FUNCTION_BLOCK FB_McAxis
VAR
  _AxisRef                      : POINTER TO Tc2_MC2.AXIS_REF;
  _pCalibrationCam              : POINTER TO BOOL;

  _nErrorId                     : UDINT; // datafield for MC error

  // MC_Power inputs for feed fwd, feed bwd, override
  _bEnablePositive              : BOOL  := TRUE;
  _bEnableNegative              : BOOL  := TRUE;
  _rAxisOverride                : LREAL := 100.0;

  _rValueParameterRead          : LREAL;
  _fbReadParameter              : Tc2_MC2.MC_ReadParameter;
  _fbWriteParameter             : Tc2_MC2.MC_WriteParameter;
  _fbWriteParameterPersist      : Tc2_MC2.MC_WriteParameterPersistent;


  // name and encoder type are read by ADSREAD instance from NC
  _sAxisName                    : STRING(30) := 'NO NAME'; // AxisName is limited to 30 chars, IdxGrp := 4000 + _AxisRef.NcToPlc.AxisId, IdxOffs := 16#02
  _sEncoderType                 : STRING(30) := 'NO TYPE';
  _nEncoderType                 : UDINT;
  _eEncoderType                 : E_AxisEncoderType;

  // Motion Control FB Instances
  _fbPower                      : Tc2_MC2.MC_Power;
  _fbReset                      : Tc2_MC2.MC_Reset;
  _fbHalt                       : Tc2_MC2.MC_Halt;
  _fbStop                       : Tc2_MC2.MC_Stop;
  _fbHome                       : Tc2_MC2.MC_Home;
  _fbJog                        : Tc2_MC2.MC_Jog;

  _fbMoveVelocity               : ARRAY[1..2]   OF  Tc2_MC2.MC_MoveVelocity;
  _fbMoveAbsolute               : ARRAY[1..2]   OF  Tc2_MC2.MC_MoveAbsolute;

  // ADS read instance for reading startup information from NC
  _fbADSRead                     : ADSREAD;

  // startup states for getting ADS information from NC
  _nStartUpErrorState,
  _nStartUp                     : DINT := 0;

  _bStartUpError,
  _bStartUp                     : BOOL;

  _rCycleTime                   : LREAL;
  _fbGetCurTaskIndex            : Tc2_System.GETCURTASKINDEX;
END_VAR

PROPERTY AxisEnableNegative : BOOL
GET
AxisEnableNegative := _bEnableNegative;
END_GET
SET
_bEnableNegative := AxisEnableNegative;
END_SET
END_PROPERTY

PROPERTY AxisEnablePositive : BOOL
GET
AxisEnablePositive  := _bEnablePositive;
END_GET
SET
_bEnablePositive := AxisEnablePositive;
END_SET
END_PROPERTY

PROPERTY AxisName : string(30)
GET
AxisName := _sAxisName;
END_GET
END_PROPERTY

PROPERTY AxisRef : pointer to Tc2_MC2.AXIS_REF
SET
_AxisRef := AxisRef;
END_SET
END_PROPERTY

PROPERTY CalibrationCam : pointer to bool
GET
CalibrationCam  := _pCalibrationCam;
END_GET
SET
_pCalibrationCam := CalibrationCam;
END_SET
END_PROPERTY

METHOD Cycle : E_PROGRESS
VAR_INST
  _eState           : E_PROGRESS;
  _rValue           : LREAL;
  _nErrorId         : UDINT;
  _stMsg            : ST_Message;
END_VAR
// call cyclic NC interface
_AxisRef^();

_fbPower(
        Axis                      := _AxisRef^, 
        Enable_Positive           := _bEnablePositive, 
        Enable_Negative           := _bEnableNegative, 
        Override                  := _rAxisOverride);

CASE _eState
OF
  E_PROGRESS.INIT:
    _fbGetCurTaskIndex();
    _rCycleTime                   := UDINT_TO_LREAL(_TaskInfo[_fbGetCurTaskIndex.index].CycleTime)/10000.0;

    _eState                       := E_PROGRESS.BUSY;
END_CASE
CASE _eState
OF
  E_PROGRESS.BUSY:
    IF (_fbPower.Error) OR
       (_AxisRef^.Status.Error)
    THEN
      _eState                     := E_PROGRESS.ERROR;

      _nErrorId                   := SEL((_fbPower.ErrorID > 0), _AxisRef^.NcToPlc.ErrorCode, _fbPower.ErrorID);

      _stMsg.eType                := E_MessageType.eMessageError;
      _stMsg.eDevice              := e_Device.Axis + TO_DINT(_AxisRef^.NcToPlc.AxisId);;
      _stMsg.eSubdevice           := e_Subdevice.fbAxis_Cycle;
      _stMsg.iErrorNumber         := _nErrorId;

      f_MessageSet(_stMsg);
    ELSE
      _nErrorId                   := 0;
      _eState                     := E_PROGRESS.WORKING;
    END_IF
END_CASE
CASE _eState
OF
  E_PROGRESS.WORKING:
    // rinse, repeat
    _eState                       := E_PROGRESS.BUSY;
    Cycle                         := E_PROGRESS.WORKING;
END_CASE
CASE _eState
OF
  E_PROGRESS.ERROR:
    IF NOT (_fbPower.Error)
    THEN
      _eState                     := E_PROGRESS.BUSY;
    ELSE
      Cycle                       := E_PROGRESS.ERROR;
    END_IF
END_CASE
END_METHOD

METHOD Disable : E_PROGRESS
VAR_INPUT
  Execute           : BOOL;
END_VAR
VAR_INST
  _eState           : E_PROGRESS;
  _rValue           : LREAL;
  _stMsg            : ST_Message;


END_VAR
IF NOT Execute THEN _eState := E_PROGRESS.INIT; END_IF

CASE _eState
OF
  E_PROGRESS.INIT:
    IF Execute 
    THEN
      memset(ADR(_stMsg),0,SIZEOF(_stMsg));
      _nErrorId                     := 0;
      _rValue                       := 0;
      _eState                       := E_PROGRESS.BUSY;
    END_IF
END_CASE
CASE _eState
OF
  E_PROGRESS.BUSY:
    _fbPower.Enable                 := FALSE;
    _eState                         := E_PROGRESS.STARTUP;
END_CASE
CASE _eState
OF
  E_PROGRESS.STARTUP:
    IF _fbPower.Error
    THEN
      _eState                       := E_PROGRESS.ERROR;
    ELSE
      _eState                       := E_PROGRESS.WAITING;
    END_IF
END_CASE
CASE _eState
OF
  E_PROGRESS.WAITING:
    IF _AxisRef^.Status.Error
    THEN
      _nErrorId                     := _AxisRef^.NcToPlc.ErrorCode;
    
      _stMsg.eType                  := E_MessageType.eMessageError;
      _stMsg.eDevice                := e_Device.Axis + TO_DINT(_AxisRef^.NcToPlc.AxisId);
      _stMsg.eSubdevice             :=  e_SubDevice.AxisControl;
      _stMsg.iErrorNumber           := _nErrorId;

      f_MessageSet(_stMsg);
    
      _eState                       := E_PROGRESS.ERROR;

    ELSIF NOT _AxisRef^.Status.ControlLoopClosed
    THEN
      _eState                       := E_PROGRESS.WORKING;
    END_IF
END_CASE
CASE _eState
OF
  E_PROGRESS.WORKING:
    _eState                         := E_PROGRESS.DONE;
END_CASE

Disable := _eState;
END_METHOD

METHOD Enable : E_PROGRESS
VAR_INPUT
  Execute           : BOOL;
END_VAR
VAR_INST
  _eState           : E_PROGRESS;
  _rValue           : LREAL;
  _stMsg            : ST_Message;
END_VAR
IF NOT Execute THEN _eState := E_PROGRESS.INIT; END_IF

CASE _eState
OF
  E_PROGRESS.INIT:
    IF Execute 
    THEN
      memset(ADR(_stMsg),0,SIZEOF(_stMsg));
      _nErrorId                     := 0;
      _rValue                       := 0;
      _eState                       := E_PROGRESS.BUSY;
    END_IF
END_CASE
CASE _eState
OF
  E_PROGRESS.BUSY:
    _fbPower.Enable                 := TRUE;
    _eState                         := E_PROGRESS.STARTUP;
END_CASE
CASE _eState
OF
  E_PROGRESS.STARTUP:
    IF _fbPower.Error
    THEN
      _fbPower.Enable               := FALSE;
      _eState                       := E_PROGRESS.ERROR;
    ELSE
      _eState                       := E_PROGRESS.WAITING;
    END_IF
END_CASE
CASE _eState
OF
  E_PROGRESS.WAITING:
    IF _AxisRef^.Status.Error
    THEN
      _nErrorId                     := _AxisRef^.NcToPlc.ErrorCode;
    
      _stMsg.eType                  := E_MessageType.eMessageError;
      _stMsg.eDevice                := e_Device.Axis + TO_DINT(_AxisRef^.NcToPlc.AxisId);
      _stMsg.eSubdevice             :=  e_SubDevice.AxisControl;
      _stMsg.iErrorNumber           := _nErrorId;
    
      f_MessageSet(_stMsg);

      _eState                       := E_PROGRESS.ERROR;

    ELSIF _AxisRef^.Status.ControlLoopClosed
    THEN
      _eState                       := E_PROGRESS.WORKING;
    END_IF
END_CASE
CASE _eState
OF
  E_PROGRESS.WORKING:
    _eState                         := E_PROGRESS.DONE;
END_CASE

Enable                              := _eState;
END_METHOD

PROPERTY EncoderType : E_AxisEncoderType
GET
EncoderType := _eEncoderType;
END_GET
END_PROPERTY

PROPERTY ErrorId : udint
GET
ErrorId := _nErrorId;
END_GET
END_PROPERTY

METHOD Halt : E_PROGRESS
VAR_INPUT
  Execute           : BOOL;
  Dec               : LREAL;
  Jerk              : LREAL;
END_VAR
VAR_INST
  _eState           : E_PROGRESS;
  _rValue           : LREAL;
  _stMsg            : ST_Message;
END_VAR
IF NOT Execute THEN _eState := E_PROGRESS.INIT; END_IF

CASE _eState
OF
  E_PROGRESS.INIT:
    IF Execute 
    THEN
      memset(ADR(_stMsg),0,SIZEOF(_stMsg));
      _nErrorId                     := 0;
      _rValue                       := 0;
      _eState                       := E_PROGRESS.BUSY;
    END_IF
END_CASE
CASE _eState
OF
  E_PROGRESS.BUSY:
    _eState                         := E_PROGRESS.WAITING;
    _fbHalt(
              Axis                  := _AxisRef^, 
              Execute               := FALSE, 
              Deceleration          := Dec, 
              Jerk                  := Jerk, 
              BufferMode            := Tc2_MC2.MC_BufferMode.MC_Aborting);
END_CASE
CASE _eState
OF
  E_PROGRESS.WAITING:
    _fbHalt(
              Axis                  := _AxisRef^, 
              Execute               := TRUE, 
              Deceleration          := Dec, 
              Jerk                  := Jerk, 
              BufferMode            := Tc2_MC2.MC_BufferMode.MC_Aborting);

    IF _fbhalt.Error
    THEN
        _nErrorId                   := _fbHalt.ErrorID;

        _stMsg.eType                := E_MessageType.eMessageError;
        _stMsg.eDevice              := e_Device.Axis + TO_DINT(_AxisRef^.NcToPlc.AxisId);
        _stMsg.eSubdevice           := e_SubDevice.fbHalt;
        _stMsg.iErrorNumber         := _nErrorId;

        f_MessageSet(_stMsg);
        _fbHalt(
              Axis                  := _AxisRef^, 
              Execute               := FALSE);

      _eState                       := E_PROGRESS.ERROR;

    ELSE
      IF _fbHalt.Done OR
         _AxisRef^.Status.NotMoving
      THEN
        _eState                     := E_PROGRESS.WORKING;

      ELSIF _fbHalt.CommandAborted
      THEN
        _eState                     := E_PROGRESS.BUSY;
      END_IF
    END_IF
END_CASE
CASE _eState
OF
  E_PROGRESS.WORKING:
    _fbHalt(
              Axis                  := _AxisRef^, 
              Execute               := FALSE);

    _eState                         := E_PROGRESS.DONE;
END_CASE

Halt := _eState;
END_METHOD

METHOD Home : E_PROGRESS
VAR_INPUT
  Execute           : BOOL;
  Position          : LREAL := DEFAULT_HOME_POSITION;
  HomingMode        : Tc2_MC2.MC_HomingMode := MC_DefaultHoming;
  Options           : Tc2_MC2.ST_HomingOptions;
END_VAR
VAR_INST
  _eState           : E_PROGRESS;
  _sValue           : STRING(40);
  _rValue           : LREAL;
  _stMsg            : ST_Message;
END_VAR
IF NOT Execute THEN _eState := E_PROGRESS.INIT; END_IF

CASE _eState
OF
  E_PROGRESS.INIT:
    IF Execute 
    THEN
      memset(ADR(_stMsg), 0,SIZEOF(_stMsg));
      memset(ADR(_sValue),0,SIZEOF(_sValue));

      _nErrorId                     := 0;
      _rValue                       := 0;
      _eState                       := E_PROGRESS.BUSY;

      IF NOT (_pCalibrationCam <> 0) 
      THEN
        // prevent page fault
        _sValue                     := 'Pointer to calibration cam not set';

        _nErrorId                   := 666;

        _stMsg.eType                := E_MessageType.eMessageError;
        _stMsg.eDevice              := e_Device.Axis + TO_DINT(_AxisRef^.NcToPlc.AxisId);
        _stMsg.eSubdevice           := e_SubDevice.fbHome;
        _stMsg.iErrorNumber         := _nErrorId;
        _stMsg.sText                := _sValue;

        f_MessageSet(_stMsg);

        _eState                     := E_PROGRESS.ERROR;
      END_IF
    END_IF
END_CASE
CASE _eState
OF
  E_PROGRESS.BUSY:
    _eState                         := E_PROGRESS.WAITING;
    _fbHome(
            Axis                    := _AxisRef^, 
            Execute                 := FALSE, 
            Position                := Position, 
            HomingMode              := HomingMode, 
            Options                 := Options, 
            bCalibrationCam         := _pCalibrationCam^);
END_CASE
CASE _eState
OF
  E_PROGRESS.WAITING:
    _fbHome(
            Execute                 := TRUE, 
            Axis                    := _AxisRef^);

    IF _fbHome.Done
    THEN
      _eState                       := E_PROGRESS.WORKING;
    ELSE
      IF _fbHome.Error
      THEN
        _eState                     := E_PROGRESS.ERROR;
        _nErrorId                   := _fbHome.ErrorID;

        _stMsg.eType                := E_MessageType.eMessageError;
        _stMsg.eDevice              := e_Device.Axis + TO_DINT(_AxisRef^.NcToPlc.AxisId);
        _stMsg.eSubdevice           :=  e_SubDevice.fbHome;
        _stMsg.iErrorNumber         := _nErrorId;

        f_MessageSet(_stMsg);

        _fbHome(
            Execute                 := FALSE, 
            Axis                    := _AxisRef^);
      END_IF
    END_IF
END_CASE
CASE _eState
OF
  E_PROGRESS.WORKING:
    _fbHome(
            Execute                 := FALSE, 
            Axis                    := _AxisRef^);

    _eState                         := E_PROGRESS.DONE;
END_CASE

Home                                := _eState;
END_METHOD

METHOD MovePosBuffer : E_PROGRESS
VAR_INPUT
  Enable          : BOOL;
  Position        : LREAL;
  Vel             : LREAL;
  Acc             : LREAL;
  Dec             : LREAL;
  Jerk            : LREAL;
  BufferMode      : Tc2_MC2.MC_BufferMode;
END_VAR
VAR_INST
  _eState           : E_PROGRESS;
  _rValue           : LREAL;
  _stMsg            : ST_Message;
END_VAR
IF NOT Enable THEN _eState := E_PROGRESS.INIT; END_IF

CASE _eState
OF
  E_PROGRESS.INIT:
    IF Enable 
    THEN
      memset(ADR(_stMsg),0,SIZEOF(_stMsg));
      _nErrorId                     := 0;
      _rValue                       := 0;
      _eState                       := E_PROGRESS.BUSY;
    END_IF
END_CASE
CASE _eState
OF
  E_PROGRESS.BUSY:
    _eState                         := E_PROGRESS.STARTUP;
    _rValue                         := Position;

    _fbMoveAbsolute[1](Axis         := _AxisRef^,
                       Execute      := FALSE);
    _fbMoveAbsolute[2](Axis         := _AxisRef^,
                       Execute      := FALSE);

END_CASE
CASE _eState
OF
  E_PROGRESS.STARTUP:
    _fbMoveAbsolute[1](
                    Axis            := _AxisRef^, 
                    Execute         := TRUE,
                    Position        := _rValue, 
                    Velocity        := Vel, 
                    Acceleration    := Acc, 
                    Deceleration    := Dec, 
                    Jerk            := Jerk, 
                    BufferMode      := BufferMode);

    _fbMoveAbsolute[2](
                    Axis            := _AxisRef^, 
                    Execute         := FALSE, 
                    Velocity        := Vel, 
                    Acceleration    := Acc, 
                    Deceleration    := Dec, 
                    Jerk            := Jerk, 
                    BufferMode      := BufferMode);

    _eState                         := E_PROGRESS.PREPARE;
END_CASE
CASE _eState
OF
  E_PROGRESS.PREPARE:
    _fbMoveAbsolute[1](Axis         := _AxisRef^);
    _fbMoveAbsolute[2](Axis         := _AxisRef^);

    IF (Position <> _rValue)
    THEN
      _rValue                       := Position;
      _eState                       := E_PROGRESS.READY;
    END_IF


END_CASE
CASE _eState
OF
  E_PROGRESS.READY:
    _fbMoveAbsolute[1](
                    Axis            := _AxisRef^, 
                    Execute         := FALSE,
                    Velocity        := Vel, 
                    Acceleration    := Acc, 
                    Deceleration    := Dec, 
                    Jerk            := Jerk, 
                    BufferMode      := BufferMode);

    _fbMoveAbsolute[2](
                    Axis            := _AxisRef^, 
                    Execute         := TRUE,
                    Position        := _rValue, 
                    Velocity        := Vel, 
                    Acceleration    := Acc, 
                    Deceleration    := Dec, 
                    Jerk            := Jerk, 
                    BufferMode      := BufferMode);
    _eState                         := E_PROGRESS.WAITING;
END_CASE
CASE _eState
OF
  E_PROGRESS.WAITING:
    _fbMoveAbsolute[1](Axis         := _AxisRef^);
    _fbMoveAbsolute[2](Axis         := _AxisRef^);

    IF (Position <> _rValue)
    THEN
      _rValue                       := Position;
      _eState                       := E_PROGRESS.STARTUP;
    END_IF
END_CASE

CASE _eState
OF
  E_PROGRESS.ERROR:
    _fbMoveAbsolute[1](Axis         := _AxisRef^,
                       Execute      := FALSE);
    _fbMoveAbsolute[2](Axis         := _AxisRef^,
                       Execute      := FALSE);

    MovePosBuffer                      := _eState;
    RETURN;
END_CASE


IF _fbMoveAbsolute[1].Error
THEN
  _nErrorId                       := _fbMoveAbsolute[1].ErrorID;

  _stMsg.eType                    := E_MessageType.eMessageError;
  _stMsg.eDevice                  := e_Device.Axis + TO_DINT(_AxisRef^.NcToPlc.AxisId);
  _stMsg.eSubdevice               :=  e_SubDevice.fbMoveAbsolute1;
  _stMsg.iErrorNumber             := _nErrorId;

  f_MessageSet(_stMsg);

  _eState                         := E_PROGRESS.ERROR;
END_IF

IF _fbMoveAbsolute[2].Error
THEN
  _nErrorId                       := _fbMoveAbsolute[2].ErrorID;

  _stMsg.eType                    := E_MessageType.eMessageError;
  _stMsg.eDevice                  := e_Device.Axis + TO_DINT(_AxisRef^.NcToPlc.AxisId);
  _stMsg.eSubdevice               :=  e_SubDevice.fbMoveAbsolute2;
  _stMsg.iErrorNumber             := _nErrorId;

  f_MessageSet(_stMsg);

  _eState                         := E_PROGRESS.ERROR;
END_IF


MovePosBuffer := _eState;
END_METHOD

METHOD MoveToPos : E_PROGRESS
VAR_INPUT
  Execute         : BOOL;
  Position        : LREAL;
  Vel             : LREAL;
  Acc             : LREAL;
  Dec             : LREAL;
  Jerk            : LREAL;
  BufferMode      : Tc2_MC2.MC_BufferMode;
END_VAR
VAR_INST
  _eState           : E_PROGRESS;
  _rValue           : LREAL;
  _rTarget          : LREAL := 0.1;
  _stMsg            : ST_Message;
END_VAR
IF NOT Execute THEN _eState := E_PROGRESS.INIT; END_IF

CASE _eState
OF
  E_PROGRESS.INIT:
    IF Execute 
    THEN
      memset(ADR(_stMsg),0,SIZEOF(_stMsg));
      _nErrorId                     := 0;
      _rValue                       := 0;
      _eState                       := E_PROGRESS.BUSY;
    END_IF
END_CASE
CASE _eState
OF
  E_PROGRESS.BUSY:
    _eState                         := E_PROGRESS.STARTUP;
    _rValue                         := Position;

    _fbMoveAbsolute[1](Axis         := _AxisRef^,
                       Execute      := FALSE);
END_CASE
CASE _eState
OF
  E_PROGRESS.STARTUP:
    _fbMoveAbsolute[1](
                    Axis            := _AxisRef^, 
                    Execute         := TRUE,
                    Position        := _rValue, 
                    Velocity        := Vel, 
                    Acceleration    := Acc, 
                    Deceleration    := Dec, 
                    Jerk            := Jerk, 
                    BufferMode      := BufferMode);

    _eState                         := E_PROGRESS.PREPARE;
END_CASE
CASE _eState
OF
  E_PROGRESS.PREPARE:
    _fbMoveAbsolute[1](Axis         := _AxisRef^);

    IF (_fbMoveAbsolute[1].Error)
    THEN
      _nErrorId                     := _fbMoveAbsolute[1].ErrorID;
    
      _stMsg.eType                  := E_MessageType.eMessageError;
      _stMsg.eDevice                := e_Device.Axis + TO_DINT(_AxisRef^.NcToPlc.AxisId);
      _stMsg.eSubdevice             :=  e_SubDevice.fbMoveAbsolute1;
      _stMsg.iErrorNumber           := _nErrorId;
    
      f_MessageSet(_stMsg);
    
      _eState                         := E_PROGRESS.ERROR;

    ELSIF (_fbMoveAbsolute[1].Active)
    THEN
      _eState                       := E_PROGRESS.WAITING;
    END_IF
END_CASE
CASE _eState
OF
  E_PROGRESS.WAITING:
    _fbMoveAbsolute[1](Axis         := _AxisRef^);

    IF (_fbMoveAbsolute[1].Error)
    THEN
      _nErrorId                     := _fbMoveAbsolute[1].ErrorID;
    
      _stMsg.eType                  := E_MessageType.eMessageError;
      _stMsg.eDevice                := e_Device.Axis + TO_DINT(_AxisRef^.NcToPlc.AxisId);
      _stMsg.eSubdevice             :=  e_SubDevice.fbMoveAbsolute1;
      _stMsg.iErrorNumber           := _nErrorId;
    
      f_MessageSet(_stMsg);
    
      _eState                         := E_PROGRESS.ERROR;

    ELSIF (_AxisRef^.Status.NotMoving) AND
       ((_AxisRef^.NcToPlc.ActPos < _fbMoveAbsolute[1].Position + _rTarget) OR
        (_AxisRef^.NcToPlc.ActPos > _fbMoveAbsolute[1].Position - _rTarget))
    THEN
      _fbMoveAbsolute[1](Axis       := _AxisRef^,
                         Execute    := FALSE);

      _eState                       := E_PROGRESS.DONE;
    END_IF
END_CASE

MoveToPos                             := _eState;
END_METHOD

METHOD MoveVelo : E_PROGRESS
VAR_INPUT
  Execute           : BOOL;
  Velocity          : LREAL;
  Acc               : LREAL;
  Dec               : LREAL;
  Jerk              : LREAL;
  Direction         : Tc2_MC2.MC_Direction := MC_Positive_Direction;
  BufferMode        : Tc2_MC2.MC_BufferMode;
END_VAR
VAR_INST
  _eState           : E_PROGRESS;
  _rValue           : LREAL;
  _stMsg            : ST_Message;
END_VAR
IF NOT Execute THEN _eState := E_PROGRESS.INIT; END_IF

CASE _eState
OF
  E_PROGRESS.INIT:
    IF Execute 
    THEN
      memset(ADR(_stMsg),0,SIZEOF(_stMsg));
      _nErrorId                     := 0;
      _rValue                       := 0;
      _eState                       := E_PROGRESS.BUSY;
    END_IF
END_CASE
CASE _eState
OF
  E_PROGRESS.BUSY:
    _eState                         := E_PROGRESS.STARTUP;
    _fbMoveVelocity[1](
                      Axis          := _AxisRef^, 
                      Execute       := FALSE, 
                      Velocity      := Velocity, 
                      Acceleration  := Acc, 
                      Deceleration  := Dec, 
                      Jerk          := Jerk, 
                      Direction     := Direction, 
                      BufferMode    := BufferMode);
END_CASE
CASE _eState
OF
  E_PROGRESS.STARTUP:
    _fbMoveVelocity[1](
                      Axis          := _AxisRef^, 
                      Execute       := TRUE);
    _eState                         := E_PROGRESS.WAITING;
END_CASE
CASE _eState
OF
  E_PROGRESS.WAITING:
    _fbMoveVelocity[1](
                      Axis          := _AxisRef^);

  IF _fbMoveVelocity[1].Error
  THEN
    _nErrorId                       := _fbMoveVelocity[1].ErrorID;
  
    _stMsg.eType                    := E_MessageType.eMessageError;
    _stMsg.eDevice                  := e_Device.Axis + TO_DINT(_AxisRef^.NcToPlc.AxisId);
    _stMsg.eSubdevice               :=  e_SubDevice.fbMoveVelocity1;
    _stMsg.iErrorNumber             := _nErrorId;
  
    f_MessageSet(_stMsg);
  
    _eState                         := E_PROGRESS.ERROR;

    ELSIF _fbMoveVelocity[1].InVelocity
    THEN
      _eState                       := E_PROGRESS.WORKING;
    END_IF
END_CASE
CASE _eState
OF
  E_PROGRESS.WORKING:
    _fbMoveVelocity[1](
                      Axis          := _AxisRef^, 
                      Execute       := FALSE);

    _eState                         := E_PROGRESS.DONE;
END_CASE


MoveVelo                            := _eState;
END_METHOD

METHOD MoveVeloBuffer : E_PROGRESS
VAR_INPUT
  Enable          : BOOL;
  Velocity        : LREAL;
  Acc             : LREAL;
  Dec             : LREAL;
  Jerk            : LREAL;
  BufferMode      : Tc2_MC2.MC_BufferMode;
END_VAR
VAR_INST
  _eState           : E_PROGRESS;
  _rValue           : LREAL;
  _stMsg            : ST_Message;
END_VAR
IF NOT Enable THEN _eState := E_PROGRESS.INIT; END_IF

CASE _eState
OF
  E_PROGRESS.INIT:
    IF Enable 
    THEN
      memset(ADR(_stMsg),0,SIZEOF(_stMsg));
      _nErrorId                     := 0;
      _rValue                       := 0;
      _eState                       := E_PROGRESS.BUSY;
    END_IF
END_CASE
CASE _eState
OF
  E_PROGRESS.BUSY:
    _eState                         := E_PROGRESS.STARTUP;
    _rValue                         := Velocity;

    _fbMoveVelocity[1](Axis         := _AxisRef^,
                       Execute      := FALSE);
    _fbMoveVelocity[2](Axis         := _AxisRef^,
                       Execute      := FALSE);

END_CASE
CASE _eState
OF
  E_PROGRESS.STARTUP:
    _fbMoveVelocity[1](
                    Axis            := _AxisRef^, 
                    Execute         := TRUE,
                    Velocity        := _rValue, 
                    Acceleration    := Acc, 
                    Deceleration    := Dec, 
                    Jerk            := Jerk, 
                    BufferMode      := BufferMode);

    _fbMoveVelocity[2](
                    Axis            := _AxisRef^, 
                    Execute         := FALSE, 
                    Acceleration    := Acc, 
                    Deceleration    := Dec, 
                    Jerk            := Jerk, 
                    BufferMode      := BufferMode);

    _eState                         := E_PROGRESS.PREPARE;
END_CASE
CASE _eState
OF
  E_PROGRESS.PREPARE:
    _fbMoveVelocity[1](Axis         := _AxisRef^);
    _fbMoveVelocity[2](Axis         := _AxisRef^);

  IF _fbMoveVelocity[1].Error
  THEN
    _nErrorId                       := _fbMoveVelocity[1].ErrorID;
  
    _stMsg.eType                    := E_MessageType.eMessageError;
    _stMsg.eDevice                  := e_Device.Axis + TO_DINT(_AxisRef^.NcToPlc.AxisId);
    _stMsg.eSubdevice               :=  e_SubDevice.fbMoveVelocity1;
    _stMsg.iErrorNumber             := _nErrorId;
  
    f_MessageSet(_stMsg);
  
    _eState                         := E_PROGRESS.ERROR;

    ELSIF (Velocity <> _rValue)
    THEN
      _rValue                       := Velocity;
      _eState                       := E_PROGRESS.READY;
    END_IF
END_CASE
CASE _eState
OF
  E_PROGRESS.READY:
    _fbMoveVelocity[1](
                    Axis            := _AxisRef^, 
                    Execute         := FALSE,
                    Acceleration    := Acc, 
                    Deceleration    := Dec, 
                    Jerk            := Jerk, 
                    BufferMode      := BufferMode);

    _fbMoveVelocity[2](
                    Axis            := _AxisRef^, 
                    Execute         := TRUE,
                    Velocity        := _rValue, 
                    Acceleration    := Acc, 
                    Deceleration    := Dec, 
                    Jerk            := Jerk, 
                    BufferMode      := BufferMode);
    _eState                         := E_PROGRESS.WAITING;
END_CASE
CASE _eState
OF
  E_PROGRESS.WAITING:
    _fbMoveVelocity[1](Axis         := _AxisRef^);
    _fbMoveVelocity[2](Axis         := _AxisRef^);

  IF _fbMoveVelocity[2].Error
  THEN
    _nErrorId                       := _fbMoveVelocity[2].ErrorID;
  
    _stMsg.eType                    := E_MessageType.eMessageError;
    _stMsg.eDevice                  := e_Device.Axis + TO_DINT(_AxisRef^.NcToPlc.AxisId);
    _stMsg.eSubdevice               :=  e_SubDevice.fbMoveVelocity2;
    _stMsg.iErrorNumber             := _nErrorId;
  
    f_MessageSet(_stMsg);
  
    _eState                         := E_PROGRESS.ERROR;

    ELSIF (Velocity <> _rValue)
    THEN
      _rValue                       := Velocity;
      _eState                       := E_PROGRESS.STARTUP;
    END_IF
END_CASE

CASE _eState
OF
  E_PROGRESS.ERROR:
    _fbMoveVelocity[1](Axis         := _AxisRef^,
                       Execute      := FALSE);
    _fbMoveVelocity[2](Axis         := _AxisRef^,
                       Execute      := FALSE);
END_CASE


MoveVeloBuffer                      := _eState;
END_METHOD

PROPERTY Override : lreal
GET
Override := _rAxisOverride;
END_GET
SET
_rAxisOverride  := Override;
END_SET
END_PROPERTY

METHOD ReadParameter : E_PROGRESS
VAR_INPUT
  Execute           : BOOL;
  ParameterNumber   : Tc2_MC2.MC_AxisParameter;
END_VAR
VAR_INST
  _eState           : E_PROGRESS;
  _rValue           : LREAL;
  _stMsg            : ST_Message;
END_VAR
IF NOT Execute THEN _eState := E_PROGRESS.INIT; END_IF

CASE _eState
OF
  E_PROGRESS.INIT:
    IF Execute 
    THEN
      memset(ADR(_stMsg),0,SIZEOF(_stMsg));
      _nErrorId                     := 0;
      _rValue                       := 0;
      _eState                       := E_PROGRESS.BUSY;
    END_IF
END_CASE
CASE _eState
OF
  E_PROGRESS.BUSY:
    _eState                         := E_PROGRESS.STARTUP;
    _fbReadParameter(
                    Axis            := _AxisRef^, 
                    Enable          := FALSE, 
                    ParameterNumber := ParameterNumber, 
                    ReadMode        := Tc2_MC2.READMODE_ONCE, 
                    Value           => _rValue);
END_CASE
CASE _eState
OF
  E_PROGRESS.STARTUP:
    _eState                         := E_PROGRESS.WAITING;
    _fbReadParameter(
                    Axis            := _AxisRef^, 
                    Enable          := TRUE, 
                    ParameterNumber := ParameterNumber, 
                    ReadMode        := Tc2_MC2.READMODE_ONCE, 
                    Value           => _rValue);
END_CASE
CASE _eState
OF
  E_PROGRESS.WAITING:
    _fbReadParameter(
                    Axis            := _AxisRef^, 
                    ParameterNumber := ParameterNumber, 
                    ReadMode        := Tc2_MC2.READMODE_ONCE, 
                    Value           => _rValue);

    IF (_fbReadParameter.Valid)
    THEN
      _rValueParameterRead          := _rValue;
      _eState                       := E_PROGRESS.WORKING;
    ELSE
      IF (_fbReadParameter.Error)
      THEN
        _nErrorId                   := _fbReadParameter.ErrorID;

        _stMsg.eType                := E_MessageType.eMessageError;
        _stMsg.eDevice              := e_Device.Axis + TO_DINT(_AxisRef^.NcToPlc.AxisId);
        _stMsg.eSubdevice           := e_SubDevice.fbReadParameter;
        _stMsg.iErrorNumber         := _nErrorId;

        f_MessageSet(_stMsg);

        _fbReadParameter(
                    Axis            := _AxisRef^, 
                    Enable          := FALSE, 
                    ParameterNumber := ParameterNumber, 
                    ReadMode        := Tc2_MC2.READMODE_ONCE, 
                    Value           => _rValue);

        _eState                     := E_PROGRESS.ERROR;
      END_IF
    END_IF
END_CASE
CASE _eState
OF
  E_PROGRESS.WORKING:
    _fbReadParameter(
                    Axis            := _AxisRef^, 
                    Enable          := FALSE, 
                    ParameterNumber := ParameterNumber, 
                    ReadMode        := Tc2_MC2.READMODE_ONCE, 
                    Value           => _rValue);

    _eState                         := E_PROGRESS.DONE;
END_CASE

ReadParameter                       := _eState;
END_METHOD

PROPERTY ReadParameterValue : LREAL
GET
ReadParameterValue := _rValueParameterRead;
END_GET
END_PROPERTY

METHOD Reset : E_PROGRESS
VAR_INPUT
  Execute           : BOOL;
END_VAR
VAR_INST
  _eState           : E_PROGRESS;
  _rValue           : LREAL;
  _stMsg            : ST_Message;
END_VAR
IF NOT Execute THEN _eState := E_PROGRESS.INIT; END_IF

CASE _eState
OF
  E_PROGRESS.INIT:
    IF Execute 
    THEN
      memset(ADR(_stMsg),0,SIZEOF(_stMsg));
      _nErrorId                   := 0;
      _rValue                     := 0;
      _eState                     := E_PROGRESS.BUSY;
    END_IF
END_CASE
CASE _eState
OF
  E_PROGRESS.BUSY:
    _eState                       := E_PROGRESS.WAITING;
    _fbReset(
              Axis                := _AxisRef^, 
              Execute             := FALSE);
END_CASE
CASE _eState
OF
  E_PROGRESS.WAITING:
    _fbReset(
              Axis                := _AxisRef^, 
              Execute             := TRUE);

    IF _fbReset.Error
    THEN
      _nErrorId                   := _fbReset.ErrorID;

      _stMsg.eType                := E_MessageType.eMessageError;
      _stMsg.eDevice              := e_Device.Axis + TO_DINT(_AxisRef^.NcToPlc.AxisId);
      _stMsg.eSubdevice           := e_SubDevice.fbReset;
      _stMsg.iErrorNumber         := _nErrorId;

      f_MessageSet(_stMsg);
      _fbReset(
              Axis                := _AxisRef^, 
              Execute             := FALSE);

      _eState                     := E_PROGRESS.ERROR;
    ELSE
      IF _fbReset.Done OR NOT
         _fbReset.Busy
      THEN
        _eState                   := E_PROGRESS.WORKING;
      END_IF
    END_IF
END_CASE
CASE _eState
OF
  E_PROGRESS.WORKING:
    _fbReset(
              Axis                := _AxisRef^, 
              Execute             := FALSE);

    _eState                       := E_PROGRESS.DONE;
END_CASE


Reset                             := _eState;
END_METHOD

METHOD SendToPos : E_PROGRESS
VAR_INPUT
  Execute         : BOOL;
  Position        : LREAL;
  Vel             : LREAL;
  Acc             : LREAL;
  Dec             : LREAL;
  Jerk            : LREAL;
  BufferMode      : Tc2_MC2.MC_BufferMode;
END_VAR
VAR_INST
  _eState           : E_PROGRESS;
  _rValue           : LREAL;
  _rTarget          : LREAL := 0.5;
  _stMsg            : ST_Message;
END_VAR
IF NOT Execute THEN _eState := E_PROGRESS.INIT; END_IF

CASE _eState
OF
  E_PROGRESS.INIT:
    IF Execute 
    THEN
      memset(ADR(_stMsg),0,SIZEOF(_stMsg));
      _nErrorId                     := 0;
      _rValue                       := 0;
      _eState                       := E_PROGRESS.BUSY;
    END_IF
END_CASE
CASE _eState
OF
  E_PROGRESS.BUSY:
    _eState                         := E_PROGRESS.STARTUP;
    _rValue                         := Position;

    _fbMoveAbsolute[1](Axis         := _AxisRef^,
                       Execute      := FALSE);
END_CASE
CASE _eState
OF
  E_PROGRESS.STARTUP:
    _fbMoveAbsolute[1](
                    Axis            := _AxisRef^, 
                    Execute         := TRUE,
                    Position        := _rValue, 
                    Velocity        := Vel, 
                    Acceleration    := Acc, 
                    Deceleration    := Dec, 
                    Jerk            := Jerk, 
                    BufferMode      := BufferMode);

    _eState                         := E_PROGRESS.PREPARE;
END_CASE
CASE _eState
OF
  E_PROGRESS.PREPARE:
    _fbMoveAbsolute[1](Axis         := _AxisRef^);

    IF (_fbMoveAbsolute[1].Error)
    THEN
      _nErrorId                     := _fbMoveAbsolute[1].ErrorID;
    
      _stMsg.eType                  := E_MessageType.eMessageError;
      _stMsg.eDevice                := e_Device.Axis + TO_DINT(_AxisRef^.NcToPlc.AxisId);
      _stMsg.eSubdevice             :=  e_SubDevice.fbMoveAbsolute1;
      _stMsg.iErrorNumber           := _nErrorId;
    
      f_MessageSet(_stMsg);
    
      _eState                         := E_PROGRESS.ERROR;

    ELSIF (_fbMoveAbsolute[1].Active)
    THEN
      _eState                       := E_PROGRESS.WAITING;
    END_IF
END_CASE
CASE _eState
OF
  E_PROGRESS.WAITING:
    _fbMoveAbsolute[1](Axis         := _AxisRef^);

    IF (_fbMoveAbsolute[1].Error)
    THEN
      _nErrorId                     := _fbMoveAbsolute[1].ErrorID;
    
      _stMsg.eType                  := E_MessageType.eMessageError;
      _stMsg.eDevice                := e_Device.Axis + TO_DINT(_AxisRef^.NcToPlc.AxisId);
      _stMsg.eSubdevice             :=  e_SubDevice.fbMoveAbsolute1;
      _stMsg.iErrorNumber           := _nErrorId;
    
      f_MessageSet(_stMsg);
    
      _eState                         := E_PROGRESS.ERROR;

    ELSIF (_AxisRef^.NcToPlc.ActPos > _fbMoveAbsolute[1].Position + _rTarget)
    THEN
      _fbMoveAbsolute[1](Axis       := _AxisRef^,
                         Execute    := FALSE);

      _eState                       := E_PROGRESS.DONE;
    END_IF
END_CASE

SendToPos                             := _eState;
END_METHOD

METHOD StartUp : E_PROGRESS
VAR_INPUT
  Execute           : BOOL;
END_VAR
VAR_INST
  _eState           : E_PROGRESS;
  _uiEncType        : UDINT;

  _sEncoder,
  _sName            : STRING(30);

  _rValue           : LREAL;
  _stMsg            : ST_Message;
END_VAR
IF NOT Execute THEN _eState := E_PROGRESS.INIT; END_IF


CASE _eState
OF
  E_PROGRESS.INIT:
    IF Execute 
    THEN
      memset(ADR(_stMsg),0,SIZEOF(_stMsg));
      _nErrorId                     := 0;
      _rValue                       := 0;
      _eState                       := E_PROGRESS.BUSY;
    END_IF
END_CASE
CASE _eState
OF
  E_PROGRESS.BUSY:
    IF (_AxisRef^.NcToPlc.AxisId <> 0)
    THEN
      _eState                       := E_PROGRESS.STARTUP;
    END_IF
END_CASE
CASE _eState
OF
  E_PROGRESS.STARTUP:
    _fbADSRead(
              NETID       := '', 
              PORT        := 501, 
              IDXGRP      := (16#5000 + _AxisRef^.NcToPlc.AxisId), 
              IDXOFFS     := 16#00000003, // offset for encoder type
              LEN         := SIZEOF(_nEncoderType), 
              DESTADDR    := ADR(_nEncoderType),
              TMOUT       := T#200MS,
              READ        := FALSE);

    // clear required ADS information
    _sAxisName      := _sName       := 'NO NAME';
    _sEncoderType   := _sEncoder    := 'NO TYPE';
    _nEncoderType   := _uiEncType   :=  0;

    _eState                         := E_PROGRESS.PREPARE;
END_CASE
CASE _eState
OF
  E_PROGRESS.PREPARE:
    _fbADSRead(
              NETID       := '', 
              PORT        := 501, 
              IDXGRP      := (16#5000 + _AxisRef^.NcToPlc.AxisId), 
              IDXOFFS     := 16#00000003, // offset for encoder type
              LEN         := SIZEOF(_nEncoderType), 
              DESTADDR    := ADR(_nEncoderType),
              TMOUT       := T#200MS,
              READ        := TRUE);

    IF (_fbADSRead.ERR)
    THEN
      _nErrorId                     := _fbAdsRead.ERRID;

      _stMsg.eType                  := E_MessageType.eMessageError;
      _stMsg.eDevice                := e_Device.Axis + TO_DINT(_AxisRef^.NcToPlc.AxisId);
      _stMsg.eSubdevice             := e_Subdevice.AxisControl;
      _stMsg.iErrorNumber           := _nErrorId;
      _stMsg.sText                  := 'StartUp Ads Error Read Encoder Type';

      f_MessageSet(_stMsg);
      _eState                       := E_PROGRESS.ERROR;

    ELSIF (_nEncoderType <> 0)
    THEN
      _uiEncType  := _eEncoderType  := _nEncoderType;
      _sEncoder   := _sEncoderType  := TO_STRING(_eEncoderType);
      _eState                       := E_PROGRESS.READY;
    END_IF
END_CASE
CASE _eState
OF
  E_PROGRESS.READY:
    _fbADSRead(
            NETID         := '', 
            PORT          := 501, 
            IDXGRP        := (16#4000 + _AxisRef^.NcToPlc.AxisId), 
            IDXOFFS       := 16#00000002, // offset for axis name
            LEN           := SIZEOF(_sAxisName), 
            DESTADDR      := ADR(_sAxisName),
            READ          := FALSE);

    _eState                         := E_PROGRESS.WAITING;
END_CASE
CASE _eState
OF
  E_PROGRESS.WAITING:
    _fbADSRead(
            NETID         := '', 
            PORT          := 501, 
            IDXGRP        := (16#4000 + _AxisRef^.NcToPlc.AxisId), 
            IDXOFFS       := 16#00000002, // offset for axis name
            LEN           := SIZEOF(_sAxisName), 
            DESTADDR      := ADR(_sAxisName),
            READ          := TRUE);

    IF (_fbADSRead.ERR)
    THEN
      _nErrorId                     := _fbAdsRead.ERRID;

      _stMsg.eType                  := E_MessageType.eMessageError;
      _stMsg.eDevice                := e_Device.Axis + TO_DINT(_AxisRef^.NcToPlc.AxisId);;
      _stMsg.eSubdevice             := e_Subdevice.AxisControl;
      _stMsg.iErrorNumber           := _nErrorId;
      _stMsg.sText                  := 'StartUp Ads Error Read Axis Name';

      f_MessageSet(_stMsg);
      _eState                       := E_PROGRESS.ERROR;

    ELSIF (_sAxisName <> 'NO NAME')
    THEN
      _sName                        := _sAxisName;
      _eState                       := E_PROGRESS.WORKING;
    END_IF
END_CASE
CASE _eState
OF
  E_PROGRESS.WORKING:
    _eState                         := E_PROGRESS.DONE;
END_CASE

StartUp                             := _eState;
END_METHOD

METHOD Stop : E_PROGRESS
VAR_INPUT
  Execute           : BOOL;
  Dec               : LREAL;
  Jerk              : LREAL;

END_VAR
VAR_INST
  _eState           : E_PROGRESS;
  _rValue           : LREAL;
  _stMsg            : ST_Message;
END_VAR
IF NOT Execute THEN _eState := E_PROGRESS.INIT; END_IF

CASE _eState
OF
  E_PROGRESS.INIT:
    IF Execute 
    THEN
      memset(ADR(_stMsg),0,SIZEOF(_stMsg));
      _nErrorId                     := 0;
      _rValue                       := 0;
      _eState                       := E_PROGRESS.BUSY;
    END_IF
END_CASE
CASE _eState
OF
  E_PROGRESS.BUSY:
    _eState                         := E_PROGRESS.WAITING;
    _fbStop(
              Axis                  := _AxisRef^, 
              Execute               := FALSE, 
              Deceleration          := Dec, 
              Jerk                  := Jerk);
END_CASE
CASE _eState
OF
  E_PROGRESS.WAITING:
    _fbStop(
              Axis                  := _AxisRef^, 
              Execute               := TRUE, 
              Deceleration          := Dec, 
              Jerk                  := Jerk);

    IF _fbStop.Error
    THEN
        _nErrorId                   := _fbStop.ErrorID;

        _stMsg.eType                := E_MessageType.eMessageError;
        _stMsg.eDevice              := e_Device.Axis + TO_DINT(_AxisRef^.NcToPlc.AxisId);
        _stMsg.eSubdevice           := e_SubDevice.fbStop;
        _stMsg.iErrorNumber         := _nErrorId;

        f_MessageSet(_stMsg);
        _fbStop(
              Axis                  := _AxisRef^, 
              Execute               := FALSE);

      _eState                       := E_PROGRESS.ERROR;

    ELSE
      IF _fbStop.Done OR
         _AxisRef^.Status.NotMoving
      THEN
        _eState                     := E_PROGRESS.WORKING;

      ELSIF _fbStop.CommandAborted
      THEN
        _eState                     := E_PROGRESS.BUSY;
      END_IF
    END_IF
END_CASE
CASE _eState
OF
  E_PROGRESS.WORKING:
    _fbStop(
              Axis                  := _AxisRef^, 
              Execute               := FALSE);

    _eState                         := E_PROGRESS.DONE;
END_CASE


Stop                                := _eState;
END_METHOD

METHOD Template : E_PROGRESS
VAR_INPUT
  Execute           : BOOL;
END_VAR
VAR_INST
  _eState           : E_PROGRESS;
  _rValue           : LREAL;
  _udiErr           : UDINT;
  _stMsg            : ST_Message;


END_VAR
IF NOT Check() THEN _eState := E_PROGRESS.ERROR; END_IF
IF NOT Execute THEN _eState := E_PROGRESS.INIT; END_IF

CASE _eState
OF
  E_PROGRESS.INIT:
    IF Execute 
    THEN
      memset(ADR(_stMsg),0,SIZEOF(_stMsg));
      _udiErr                       := 0;
      _rValue                       := 0;
      _eState                       := E_PROGRESS.BUSY;
    END_IF
END_CASE
CASE _eState
OF
  E_PROGRESS.BUSY:
    _eState                         := E_PROGRESS.STARTUP;
END_CASE
CASE _eState
OF
  E_PROGRESS.STARTUP:
    _eState                       := E_PROGRESS.PREPARE;
END_CASE
CASE _eState
OF
  E_PROGRESS.PREPARE:
    _eState                         := E_PROGRESS.READY;
END_CASE
CASE _eState
OF
  E_PROGRESS.READY:
    _eState                         := E_PROGRESS.WAITING;
END_CASE
CASE _eState
OF
  E_PROGRESS.WAITING:
    _eState                         := E_PROGRESS.WORKING;
END_CASE
CASE _eState
OF
  E_PROGRESS.WORKING:
    _eState                         := E_PROGRESS.DONE;
END_CASE

Template_1 := _eState;
END_METHOD

METHOD WriteParameter : E_PROGRESS
VAR_INPUT
  Execute           : BOOL;
  Value             : LREAL;
  ParameterNumber   : Tc2_MC2.MC_AxisParameter;
END_VAR
VAR_INST
  _eState           : E_PROGRESS;
  _nParameter       : Tc2_MC2.MC_AxisParameter;
  _rValue           : LREAL;
  _stMsg            : ST_Message;
END_VAR
IF NOT Execute THEN _eState := E_PROGRESS.INIT; END_IF

CASE _eState
OF
  E_PROGRESS.INIT:
    IF Execute 
    THEN
      memset(ADR(_stMsg),0,SIZEOF(_stMsg));
      _nParameter                   := 0;
      _nErrorId                     := 0;
      _rValue                       := 0;
      _eState                       := E_PROGRESS.BUSY;
    END_IF
END_CASE
CASE _eState
OF
  E_PROGRESS.BUSY:
    _eState                         := E_PROGRESS.STARTUP;
    _nParameter                     := ParameterNumber;

    _fbWriteParameter(
                    Axis            := _AxisRef^, 
                    Execute         := FALSE, 
                    ParameterNumber := ParameterNumber, 
                    Value           := Value);
END_CASE
CASE _eState
OF
  E_PROGRESS.STARTUP:
    _eState                         := E_PROGRESS.WAITING;
    _fbWriteParameter(
                    Axis            := _AxisRef^, 
                    Execute         := TRUE, 
                    ParameterNumber := ParameterNumber, 
                    Value           := Value);

END_CASE
CASE _eState
OF
  E_PROGRESS.WAITING:
    _fbWriteParameter(
                    Axis            := _AxisRef^, 
                    ParameterNumber := ParameterNumber, 
                    Value           := Value);

    IF _fbWriteParameter.Error
    THEN
      _nErrorId                     := _fbWriteParameter.ErrorID;

      _stMsg.eType                  := E_MessageType.eMessageError;
      _stMsg.eDevice                := e_Device.Axis + TO_DINT(_AxisRef^.NcToPlc.AxisId);
      _stMsg.eSubdevice             := e_SubDevice.fbWriteParameter;
      _stMsg.iErrorNumber           := _nErrorId;

      f_MessageSet(_stMsg);

      _fbWriteParameter(
                    Axis            := _AxisRef^,
                    Execute         := FALSE, 
                    ParameterNumber := ParameterNumber, 
                    Value           := Value);


      _eState                       := E_PROGRESS.ERROR;
    ELSE
      IF _fbWriteParameter.Done
      THEN
        _rValue                     := _fbWriteParameter.Value;
        _eState                     := E_PROGRESS.WORKING;
      END_IF
    END_IF

END_CASE
CASE _eState
OF
  E_PROGRESS.WORKING:
    _fbWriteParameter(
                    Axis            := _AxisRef^,
                    Execute         := FALSE, 
                    ParameterNumber := ParameterNumber, 
                    Value           := Value);
    _eState                         := E_PROGRESS.DONE;
END_CASE


WriteParameter                      := _eState;
END_METHOD

METHOD WriteParameterPersistent : E_PROGRESS
VAR_INPUT
  Execute           : BOOL;
  Value             : LREAL;
  ParameterNumber   : Tc2_MC2.MC_AxisParameter;
END_VAR
VAR_INST
  _eState           : E_PROGRESS;
  _rValue           : LREAL;
  _stMsg            : ST_Message;
END_VAR
IF NOT Execute THEN _eState := E_PROGRESS.INIT; END_IF

CASE _eState
OF
  E_PROGRESS.INIT:
    IF Execute 
    THEN
      memset(ADR(_stMsg),0,SIZEOF(_stMsg));
      _nErrorId                     := 0;
      _rValue                       := 0;
      _eState                       := E_PROGRESS.BUSY;
    END_IF
END_CASE
CASE _eState
OF
  E_PROGRESS.BUSY:
    _eState                         := E_PROGRESS.STARTUP;
    _fbWriteParameterPersist(
                    Axis            := _AxisRef^, 
                    Execute         := FALSE, 
                    ParameterNumber := ParameterNumber, 
                    Value           := Value);
END_CASE
CASE _eState
OF
  E_PROGRESS.STARTUP:
    _eState                         := E_PROGRESS.WAITING;
    _fbWriteParameterPersist(
                    Axis            := _AxisRef^, 
                    Execute         := TRUE, 
                    ParameterNumber := ParameterNumber, 
                    Value           := Value);

END_CASE
CASE _eState
OF
  E_PROGRESS.WAITING:
    _fbWriteParameterPersist(
                    Axis            := _AxisRef^, 
                    ParameterNumber := ParameterNumber, 
                    Value           := Value);

    IF (_fbWriteParameterPersist.Error)
    THEN
      _nErrorId                     := _fbWriteParameterPersist.ErrorID;

      _stMsg.eType                  := E_MessageType.eMessageError;
      _stMsg.eDevice                := e_Device.Axis + TO_DINT(_AxisRef^.NcToPlc.AxisId);
      _stMsg.eSubdevice             := e_SubDevice.fbWriteParameterPersistent;
      _stMsg.iErrorNumber           := _nErrorId;

      f_MessageSet(_stMsg);

      _fbWriteParameterPersist(
                    Axis            := _AxisRef^,
                    Execute         := FALSE, 
                    ParameterNumber := ParameterNumber, 
                    Value           := Value);


      _eState                       := E_PROGRESS.ERROR;
    ELSE
      IF (_fbWriteParameterPersist.Done)
      THEN
        _rValue                     := _fbWriteParameterPersist.Value;
        _eState                     := E_PROGRESS.WORKING;
      END_IF
    END_IF

END_CASE
CASE _eState
OF
  E_PROGRESS.WORKING:
    _fbWriteParameterPersist(
                    Axis            := _AxisRef^,
                    Execute         := FALSE, 
                    ParameterNumber := ParameterNumber, 
                    Value           := Value);

    _eState                         := E_PROGRESS.DONE;
END_CASE


WriteParameterPersistent            := _eState;
END_METHOD

END_FUNCTION_BLOCK

(* stored: Version 1.1.0.1, ProductVersion 3.1.4024.12
   POU FB_McAxis: Id {b0a70715-8745-098e-33e9-cc5f7a367c73}, SpecialFunc None
   Folder methods: Id {e674326e-ed43-01be-1a84-509d9487c148}
   Folder properties: Id {cb335709-3f53-0ca8-0342-0b6d016a56bb}
   Property AxisEnableNegative: Id {a1aa2814-ef28-0b58-2918-1095fb38fbbe}
   Get Get: Id {2af4d04a-c67a-0989-0200-972cb088feaa}
   Set Set: Id {f9b48d43-b5cb-0581-30cb-023409850de3}
   Property AxisEnablePositive: Id {b1ddc089-3b48-0a11-313d-0f16e9587698}
   Get Get: Id {86716297-6c0c-06d5-366c-d174b317d66e}
   Set Set: Id {4580af82-6f3c-0113-02a4-7daaef9bed88}
   Property AxisName: Id {dcc452a2-d3f9-0f06-025b-2034aaea8e70}
   Get Get: Id {da0dc137-e936-0ab7-18eb-4dd0376e1850}
   Property AxisRef: Id {d622fbfb-1430-047a-062d-a4dac266c76c}
   Set Set: Id {e30bf9e1-a426-000b-02a7-42821d5e2114}
   Property CalibrationCam: Id {2999b136-e7f2-0ed9-32d9-2c41cd4633ce}
   Get Get: Id {771a5d1e-5ee2-0432-1264-29cbfd640c0b}
   Set Set: Id {73d29774-cb40-02b1-1e9f-252b3b3d0c30}
   Method Cycle: Id {0952ac4a-b64d-0779-0df8-f45840c5c7eb}
   Method Disable: Id {3cfd1816-2e58-0ba6-30c2-feff57d138a8}
   Method Enable: Id {d3ecb8f6-2a8a-08cc-230d-f8b28d0b2674}
   Property EncoderType: Id {dd9d7c97-af96-007b-0caa-e74acc85ce7f}
   Get Get: Id {67c78f5d-4012-0b7e-3910-20eadd409eb3}
   Property ErrorId: Id {d56c7e0e-35a6-0639-16b7-19f40aaa065b}
   Get Get: Id {0b923b10-f0c2-0676-20bc-0da42dc2410d}
   Method Halt: Id {ddc30265-22a2-0ad6-2ef2-c12a5a7121f8}
   Method Home: Id {9f6b266a-70b1-05d8-2838-695e2d6a6f25}
   Method MovePosBuffer: Id {c85dc519-a612-0a41-1a3d-8c9a1d3f1397}
   Method MoveToPos: Id {9983f17a-1ed1-0daf-01b6-9e9adfd03ef3}
   Method MoveVelo: Id {f336fcbe-ff7a-0e9f-3cdd-2eac3cc75bff}
   Method MoveVeloBuffer: Id {6580e262-5fae-068b-31a4-0bea4fa7cdc2}
   Property Override: Id {2326350f-5459-0a6c-2ba9-357e1bba98f9}
   Get Get: Id {59a4c2b8-06cc-055c-2e8c-b8c096b86326}
   Set Set: Id {c4343645-132c-03c0-251d-edf786107745}
   Method ReadParameter: Id {54a806b1-3430-0c86-070c-bd7f0cce9548}
   Property ReadParameterValue: Id {5737dfc7-f28d-04d5-1795-84a65134e1c4}
   Get Get: Id {29aee24e-4dd3-0b0e-0d0c-20dcb7cad526}
   Method Reset: Id {c56fedee-350d-09ff-3f42-160d961f4e86}
   Method SendToPos: Id {897e9d2e-a3c2-006b-03c5-193d76055ec3}
   Method StartUp: Id {914834b0-e73e-0894-3b5e-bf530799f619}
   Method Stop: Id {789b9c2b-f93d-0b61-11f2-dc8daaed9df3}
   Method Template: Id {cdf187ab-3940-086d-05f1-b21d6093dcd8}
   Method WriteParameter: Id {d9084bfe-9c42-03ce-187a-0d3ac44cc9cd}
   Method WriteParameterPersistent: Id {6dcff98d-915b-08be-0870-0135f1dea9d3} *)
